# EPICS autosave request: iocs/ur-robot/ur-robot-ioc/db/rtde_io_settings.req
# Port of urRobotApp/Db/rtde_io_settings.req.
$(P)IO:SpeedSlider.VAL
